% RSLogix 500 project I2P JOB 16_RUSSELL_BAK008.RSS, saved by version 10.00.00.00 %
PROJECT "ML02A"    % processor: Bul.1763 MicroLogix 1100 Series B %

PROGRAM FILES
  LAD 2   5 rungs

DATA FILES
  O0 OUTPUT  4 elements
  I1 INPUT  6 elements
  S2 STATUS  66 elements
  B3 BINARY  1 elements
  T4 TIMER  1 elements
  C5 COUNTER  1 elements
  R6 CONTROL  1 elements
  N7 INTEGER  1 elements
  F8 FLOAT  1 elements

LADDER 2
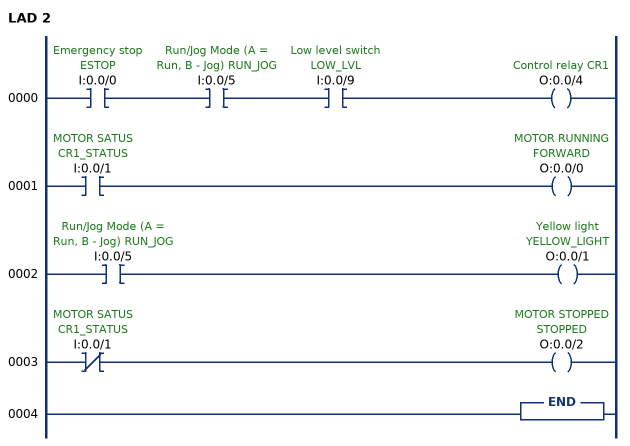
% Rung: 0 %
SOR XIC I:0.0/0 XIC I:0.0/5 XIC I:0.0/9 OTE O:0.0/4 EOR
%   I:0.0/0  ESTOP  "Emergency stop" %
%   I:0.0/5  RUN_JOG  "Run/Jog Mode (A = Run, B - Jog)" %
%   I:0.0/9  LOW_LVL  "Low level switch" %
%   O:0.0/4  CR1  "Control relay" %
% Rung: 1 %
SOR XIC I:0.0/1 OTE O:0.0/0 EOR
%   I:0.0/1  CR1_STATUS  "MOTOR SATUS" %
%   O:0.0/0  FORWARD  "MOTOR RUNNING" %
% Rung: 2 %
SOR XIC I:0.0/5 OTE O:0.0/1 EOR
%   I:0.0/5  RUN_JOG  "Run/Jog Mode (A = Run, B - Jog)" %
%   O:0.0/1  YELLOW_LIGHT  "Yellow light" %
% Rung: 3 %
SOR XIO I:0.0/1 OTE O:0.0/2 EOR
%   I:0.0/1  CR1_STATUS  "MOTOR SATUS" %
%   O:0.0/2  STOPPED  "MOTOR STOPPED" %
% Rung: 4 %
SOR END EOR

OTHER DOCUMENTED ADDRESSES
  B3:0/0  "FWD BIT"
  B3:0/1  "REV BIT"
  B3:0/2  LAST_REV
  B3:1  LAST_FWD
  I:0.0/2  CR2_STATUS  "Status of control relay 2"
  I:0.0/3  3PSS_A  "3 position selector switch A position"
  I:0.0/4  3PSS_B  "3 position selector switch B position"
  I:0.0/6  STOP  "Normally closed pushbutton"
  I:0.0/7  START  "Normally open pushbutton"
  I:0.0/8  JOG  "Normally open pushbutton"
  O:0.0/3  REVERSE  "MOTOR RUNNING"
  O:0.0/5  CR2  "Contro relay 2"

DATA TABLE (non-zero values as saved)
DATA T4
% .PRE .ACC %
% T4:0 % 32767 0
DATA C5
% .PRE .ACC %
% C5:0 % 16 8
